(*
SPDX-FileCopyrightText: © 2026 Oleksandr Tiutyk <trofimich@gmail.com>
SPDX-License-Identifier: MIT
License: https://opensource.org/license/mit
*)

INTERFACE ITrySetLightActionDescriptor EXTENDS TOF_Core.INamed

{attribute 'monitoring' := 'call'}
PROPERTY FINAL NewColor : TRAFFIC_LIGHT_COLOR
GET
END_GET
SET
END_SET
END_PROPERTY

END_INTERFACE

(* stored: Version 1.1.0.1
   Itf ITrySetLightActionDescriptor: Id {352691e8-b5a9-44d9-944a-10f3825573bc}
   Property NewColor: Id {26da345c-818e-4556-b29a-850ffe3b37ed}
   Get Get: Id {95cabc4b-fd0b-4c5c-ba03-e1540855287c}
   Set Set: Id {b9c55274-04f7-4104-b382-f5351263e3b2} *)
